FUNCTION_BLOCK EcMasterGetDeviceId IMPLEMENTS IEcTask
VAR_INPUT
END_VAR
VAR_OUTPUT
END_VAR
VAR
	iState : INT;
	getDeviceIdentity : Tc2_EtherCAT.FB_EcGetSlaveIdentity;
	_execute: BOOL;
	_done: BOOL;
	_busy: BOOL;
	_error: BOOL;
	_netId: AMSNETID;
END_VAR

CASE iState OF
	0:
		IF _execute THEN
			_done := FALSE;
			_busy := TRUE;
			_error := FALSE;
			getDeviceIdentity.bExecute := TRUE;
			IF getDeviceIdentity.bBusy THEN
				iState := 10;
				_execute := false;
			END_IF
		END_IF
	10:
		IF NOT getDeviceIdentity.bBusy THEN
			IF NOT getDeviceIdentity.bError THEN
				_done := TRUE;
			ELSE
				_error := TRUE;
			END_IF
			_busy := FALSE;
			getDeviceIdentity.bExecute := FALSE;
			iState := 0;
		END_IF
END_CASE

getDeviceIdentity(sNetId := Tc2_System.F_CreateAmsNetId(nIds := NetId));

{warning 'add method implementation '}
METHOD Abort : BOOL
getDeviceIdentity.bExecute := FALSE;
_busy := FALSE;
_execute := FALSE;
Abort := TRUE;
iState := 0;
END_METHOD

{warning 'add property implementation'}
PROPERTY Busy : BOOL
GET
Busy := _busy;
END_GET
END_PROPERTY

PROPERTY DeviceAddr : uint
GET
DeviceAddr := getDeviceIdentity.nSlaveAddr;
END_GET
SET
getDeviceIdentity.nSlaveAddr := DeviceAddr;
END_SET
END_PROPERTY

PROPERTY DeviceIdentity : ST_EcSlaveIdentity
GET
DeviceIdentity := getDeviceIdentity.identity;
END_GET
END_PROPERTY

{warning 'add property implementation'}
PROPERTY Done : BOOL
GET
Done := _done;
END_GET
END_PROPERTY

{warning 'add property implementation'}
PROPERTY Error : BOOL
GET
Error := _error;
END_GET
END_PROPERTY

{warning 'add method implementation '}
METHOD Execute : BOOL
IF NOT getDeviceIdentity.bBusy THEN
	Execute := _execute := true;
END_IF
END_METHOD

{warning 'add property implementation'}
PROPERTY NetID : amsnetid
GET
NetID := _netId;
END_GET
SET
_netId := NetID;
END_SET
END_PROPERTY

END_FUNCTION_BLOCK

(* stored: Version 1.1.0.1, ProductVersion 3.1.4024.11
   POU EcMasterGetDeviceId: Id {024e3e34-01f0-4d80-8995-7a19e9695f4b}, SpecialFunc None
   Method Abort: Id {05cae8df-dfc8-445a-9b47-a924a01974dc}
   Property Busy: Id {49b9a255-6e51-4c52-b644-dc6f0568843b}
   Get Get: Id {536b3ce0-a600-4c08-8627-d94d18b0412b}
   Property DeviceAddr: Id {e63ca9e3-be83-4948-8357-0e51909926f8}
   Get Get: Id {637e7f4e-4ec9-48fa-9a8c-bb715ff99f6e}
   Set Set: Id {7ca995c2-22e5-4bf7-be6c-b734a987e5de}
   Property DeviceIdentity: Id {dc2a1a76-84ed-469f-a25b-1f1abed482fa}
   Get Get: Id {99336325-399f-4cd2-83e2-d05d03ff692e}
   Property Done: Id {db205210-65b5-481a-a693-2482d85425c1}
   Get Get: Id {b09677dc-ad54-4dcc-b87e-e02142256212}
   Property Error: Id {8285cd50-96f2-45d9-a1de-35db29fbc19b}
   Get Get: Id {c20fb7a8-61d2-4ff6-b9e5-28608a7cac03}
   Method Execute: Id {872eb657-c2d0-42e0-ae9b-67c1a6940297}
   Property NetID: Id {d844a922-4626-49ee-83da-763d5b0355c1}
   Get Get: Id {6f8ed4f9-1745-4473-8514-e10cc7f040a1}
   Set Set: Id {50cfca93-f1bd-47c8-9149-f2f831fba509} *)
